// TwinCAT 3 PLC project Example
// ProgramVersion: 3.1.4024.0
// libraries:
//   Tc2_EtherCAT, * (Beckhoff Automation GmbH)
//   Tc2_MC2, * (Beckhoff Automation GmbH)
//   Tc2_Standard, * (Beckhoff Automation GmbH)
//   Tc2_System, * (Beckhoff Automation GmbH)
//   Tc2_Utilities, * (Beckhoff Automation GmbH)
//   Tc3_Component, * (Zerlauth)
//   Tc3_JsonXml, * (Beckhoff Automation GmbH)
//   Tc3_Module, * (Beckhoff Automation GmbH)
// project tree:
//   GVLs/ M001.TcGVL
//   InDevelopment/Axis/ FB_McAxis.TcPOU (not stored), I_Axis.TcIO (not stored)
//   InDevelopment/Ethercat/ FB_Ethercat.TcPOU
//   InDevelopment/ FB_ComponentEX.TcPOU, FB_Dictionary.TcPOU, FB_Module01.TcPOU, FB_ModuleLogger.TcPOU (not stored)
//   / PlcTask.TcTTO
//   POUs/ MAIN.TcPOU
// real-time tasks:
//   TASK PlcTask: cycle T#100000us, priority 21, ADS port 351

CONFIGURATION Example
    RESOURCE PLC ON TwinCAT3
        TASK PlcTask(INTERVAL := T#100000us, PRIORITY := 21);
        PROGRAM MAIN WITH PlcTask : MAIN;
    END_RESOURCE
END_CONFIGURATION

// ---- GVLs/M001.TcGVL
{attribute 'qualified_only'}
VAR_GLOBAL
END_VAR

// ---- POUs/MAIN.TcPOU
PROGRAM MAIN
VAR
	fbDictionary:		FB_Dictionary;
	fbEthercat:			FB_Ethercat;
	fbComponent:		FB_Module01;
	
	bReset:			BOOL;
	bStart: 		BOOL;
    bHold:       	BOOL;
    bPause:    		BOOL;
	bStop:       	BOOL;
    bAbort:      	BOOL;

	sValue: STRING(255);
END_VAR

fbDictionary();

fbDictionary.M_Add('Test', 'Value');

sValue:= fbDictionary.M_GetSTRING('Test');

fbLogger();
fbEthercat.M_Cycle();
fbComponent.M_Cycle();


IF bReset THEN
	bReset:= NOT fbComponent.M_Request(E_Request.Reset);
END_IF

IF bStart THEN
	bStart:= NOT fbComponent.M_Request(E_Request.Start);
END_IF

IF bStop THEN
	bStop:= not fbComponent.M_Request(E_Request.Stop);
END_IF

IF bHold THEN
	bHold:= NOT fbComponent.M_Request(E_Request.Hold);
END_IF

IF bPause THEN
	bPause:= NOT fbComponent.M_Request(E_Request.Pause);
END_IF

IF bAbort THEN
	bAbort:= NOT fbComponent.M_Request(E_Request.Abort);
END_IF

END_PROGRAM

// ---- InDevelopment/FB_Dictionary.TcPOU
FUNCTION_BLOCK FB_Dictionary IMPLEMENTS I_Dictionary
VAR_INPUT
END_VAR
VAR_OUTPUT
END_VAR
VAR
	bAdd:				BOOL;
	bReset:				Bool;
	bLoad:				BOOL;
	bSave:				BOOL;
	fbJson:				FB_JsonDomParser;
  	json:				SJsonValue;

	sJson: 				STRING(255);
END_VAR

IF bReset THEN
	bReset:= FALSE;
	json:= fbJson.NewDocument();
	bSave:= TRUE;
END_IF

IF bAdd THEN
	IF fbJson.FindMember(json, 'member:Value1') = 0 THEN
		fbJson.AddStringMember(json, 'member/Value1', 'Value');		
	END_IF
	IF fbJson.FindMember(json, 'member/Value2') = 0 THEN
		fbJson.AddStringMember(json, 'member/Value2', 'Value');		
	END_IF
END_IF


IF bLoad THEN
	fbJson.LoadDocumentFromFile('C:\Test.json', bLoad);
END_IF
IF bSave THEN
	fbJson.SaveDocumentToFile('C:\Test.json', bSave);
END_IF

fbJson.CopyDocument(sJson, SIZEOF(sJson));

METHOD PUBLIC M_Add : BOOL
VAR_INPUT
	Key:		STRING(255);
	Value:		STRING(255);
END_VAR
END_METHOD

METHOD PUBLIC M_GetSTRING : String(255)
VAR_INPUT
	sName:	STRING(255);
END_VAR
END_METHOD

METHOD PUBLIC M_Load : BOOL
VAR_INPUT
	sFile:	STRING(255);
END_VAR
END_METHOD

METHOD PUBLIC M_Reset : BOOL
VAR_INPUT
END_VAR
END_METHOD

METHOD PUBLIC M_Save : BOOL
VAR_INPUT
END_VAR
END_METHOD

END_FUNCTION_BLOCK

// ---- InDevelopment/Ethercat/FB_Ethercat.TcPOU
FUNCTION_BLOCK FB_Ethercat EXTENDS FB_Component
VAR_INPUT
    NetId 			AT %I*:		T_AmsNetIdArr;
	Slaves			AT %I*: 	UINT;
END_VAR
VAR_OUTPUT
END_VAR
VAR
	fbGetMasterState: 			FB_EcGetMasterDevState;
	fbMasterFrameStatistic:		FB_EcMasterFrameStatistic;
	fbGetSlaveStates:			FB_EcGetAllSlaveStates;
	pSlaveState:				POINTER TO Tc2_EtherCAT.ST_EcSlaveState;
END_VAR

METHOD PUBLIC M_Call
VAR_INPUT
END_VAR
SUPER^.M_Call();

fbGetMasterState(sNetId:= F_CreateAmsNetId(NetId));

fbMasterFrameStatistic(sNetId:= F_CreateAmsNetId(NetId));


IF pSlaveState = 0 THEN
		pSlaveState:= __NEW(BYTE, (SIZEOF(Tc2_EtherCAT.ST_EcSlaveState) * Slaves));
END_IF

fbGetSlaveStates(	sNetId:= F_CreateAmsNetId(NetId), 
					pStateBuf:= pSlaveState, 
					cbBufLen:= Slaves * SIZEOF(Tc2_EtherCAT.ST_EcSlaveState));
END_METHOD

END_FUNCTION_BLOCK

// ---- InDevelopment/FB_Module01.TcPOU
FUNCTION_BLOCK FB_Module01 EXTENDS FB_Module
VAR_INPUT
END_VAR
VAR_OUTPUT
END_VAR
VAR
	fbComponent1:				FB_Component;
	fbComponent2:				FB_Component;
	fbComponent3:				FB_ComponentEx;
	fbComponent4:				FB_ComponentChild;
END_VAR

METHOD PUBLIC M_Cylic
VAR_INPUT
END_VAR
SUPER^.M_Cylic();

fbComponent1.M_Cylic();
fbComponent2.M_Cylic();
fbComponent3.M_Cylic();
fbComponent4.M_Cylic();
END_METHOD

METHOD PROTECTED M_Execute : bool
VAR_INPUT
END_VAR
M_Execute:= SUPER^.M_Execute();

//fbEvent.M_Warning('My first Warning', '' );	
fbEvent.M_Warning('My secound Warning', '' );
END_METHOD

METHOD PROTECTED M_Initialise
VAR_INPUT
END_VAR
SUPER^.M_Initialise();
M_Attach(fbComponent1);
M_Attach(fbComponent2);
M_Attach(fbComponent3);
M_Attach(fbComponent4);
END_METHOD

METHOD PROTECTED M_Running
VAR_INPUT
END_VAR
//IF NOT M001.fbEmStop.P_Value THEN
//	fbEvent.M_AddSTRING(M001.fbEmStop.P_ID);
//	fbEvent.M_Abort('Emergency stop not ok', '');
//ELSIF NOT M001.fbPowerOn.P_Value THEN
//	fbEvent.M_AddSTRING(M001.fbPowerOn.P_ID);
//	fbEvent.M_Abort('Power not on', '');
//ELSIF NOT M001.fbFuse1.P_Value THEN
//	fbEvent.M_AddSTRING(M001.fbFuse1.P_ID);
//	fbEvent.M_Stop('Fuse Triped', '');	
	
//END_IF
END_METHOD

END_FUNCTION_BLOCK

// ---- InDevelopment/FB_ComponentEX.TcPOU
FUNCTION_BLOCK FB_ComponentEX EXTENDS FB_Component
VAR_INPUT
END_VAR
VAR_OUTPUT
END_VAR
VAR
	bAbort:			BOOL;
	bStop:			BOOL;
	bStopCycle:		BOOL;
END_VAR

METHOD PROTECTED M_Execute : BOOL
VAR_INPUT
END_VAR

IF bAbort THEN
	bAbort:= FALSE;
	fbEvent.M_AddSTRING('Test');
	fbEvent.M_AddSTRING('Test2');
	fbEvent.M_AddSTRING('Test3');
	fbEvent.M_Abort('First Error Abort', 'a');
END_IF

IF bStop THEN
	bStop:= FALSE;
	fbEvent.M_AddSTRING('Test');
	fbEvent.M_AddSTRING('Test2');
	fbEvent.M_AddSTRING('Test3');
	fbEvent.M_Stop('First Error Stop', 'b');
END_IF

IF bStopCycle THEN
	fbEvent.M_AddSTRING('Test');
	fbEvent.M_AddSTRING('Test2');
	fbEvent.M_AddSTRING('Test3');
	fbEvent.M_StopCycle('First Error Complete', 'b');
END_IF

M_Execute:= NOT bStopCycle;
END_METHOD

END_FUNCTION_BLOCK
